FUNCTION f_MoverPositionAssignementToString : string(30)
VAR_INPUT
  nPosAssignement   : UINT;
END_VAR
VAR
END_VAR


CASE nPosAssignement
OF
  0:
    f_MoverPositionAssignementToString    := 'Standard';
  1:
    f_MoverPositionAssignementToString    := 'Start At First Mover';
ELSE
    f_MoverPositionAssignementToString    := 'UNKNOWN Assignement';
END_CASE

END_FUNCTION

(* stored: Version 1.1.0.1, ProductVersion 3.1.4024.12
   POU f_MoverPositionAssignementToString: Id {b7721be6-7f52-461c-82f7-e7a956a932d5}, SpecialFunc None *)
